INTERFACE I_Stoppable EXTENDS I_Base

METHOD Stop
VAR_INPUT
END_VAR
END_METHOD

{attribute 'monitoring' := 'call'}
PROPERTY Stopped : BOOL
GET
END_GET
END_PROPERTY

END_INTERFACE

(* stored: Version 1.1.0.1, ProductVersion 3.1.4026.18
   Itf I_Stoppable: Id {a9962047-8cfb-4854-a605-5df427da7e84}
   Method Stop: Id {5a2f1397-c7f4-4baf-b67c-e98b024e4f99}
   Property Stopped: Id {10c93345-0e51-4082-90bd-feabf08dacb5}
   Get Get: Id {ce9c8dbb-92c8-47e0-b477-0958c099cea9} *)
